Universal Robots PolyScope program: lmao.urp

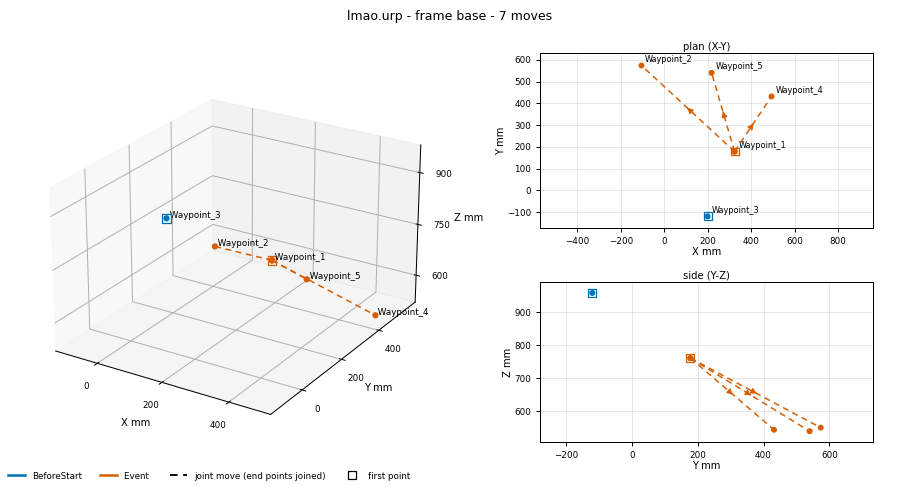
[picture p0: tool path of lmao.urp in frame base, 7 of 13 moves have a stored position in this frame; points joined in program order, loops and branches not executed]
Program lmao (createdIn=3.4.4.412 lastSavedIn=3.4.4.412 directory=/programs installation=default robotSerialNumber=2017356443)
Calibrated DH parameters: a=[0.000092, -0.116521, -0.182101, -0.000106, 0.000044, 0]; d=[0.089391, 255.189113, -82.629387, -172.449369, 0.094782, 0.082637]; alpha=[1.569598, 0.001603, 0.002015, 1.570234, -1.570307, 0]; deltaTheta=[-0.000017, 1.293309, -0.204843, -1.088417, 0.000036, -0.000078]
BeforeStart
  MoveJ speed 60 deg/s, acceleration 80 deg/s^2 (useActiveTCP=false)
    Waypoint Waypoint_3: TCP in base x=199.454 y=-120.02 z=959.051 mm, rx=-1.3734 ry=1.2247 rz=-1.3143 rad; joints [-2.468, -84.062, -29.689, -71.089, 89.859, -9.367] deg; flange x=199.397 y=-120.02 z=959.077 mm, rx=-1.3733 ry=1.2246 rz=-1.3144 rad
    URCap Gripper (Robotiq_2-Finger_Adaptive_Gripper, Robotiq Inc.) data=position = 0
      | force = 0
      | speed = 0
      | blocking = true
      | slaveIds = [9]
Robot Program (runOnlyOnce=false motionType=MoveJ speed=1.047198 acceleration=1.396263 useActiveTCP=false)
  knob := 1
  MoveJ speed 60 deg/s, acceleration 80 deg/s^2 (useActiveTCP=false)
    Waypoint Waypoint (Variable): variable(featureName=robopoint)
